PROGRAM MAIN
VAR
	bEna : BOOL;
	bbbhei : BOOL;
END_VAR

bEna := GVL.start_Button;

END_PROGRAM

(* stored: Version 1.1.0.1, ProductVersion 3.1.4024.12
   POU MAIN: Id {bf80d31d-77d1-4e56-870a-cac5c21793c4}, SpecialFunc None *)
